INTERFACE I_QuantityINT EXTENDS I_Quantity


METHOD Equals : BOOL
VAR_INPUT
    Quantity : I_QuantityINT;
END_VAR
END_METHOD


PROPERTY Val : INT
GET
END_GET
END_PROPERTY

END_INTERFACE

(* stored: Version 1.1.0.1
   Itf I_QuantityINT: Id {52fcf1d4-4739-4a46-a8fa-247f0cf96327}
   Method Equals: Id {75922ae9-885c-4929-8e5f-49b17d0821f4}
   Property Val: Id {557475ef-ad12-4e0b-9044-e63f1495b352}
   Get Get: Id {de7ee6ba-6ebc-4c25-8507-7b869ba00b61} *)
